DATA_BLOCK DB 811
TITLE =
AUTHOR : CB
STRUCT
WORD0 : WORD;	//
WORD1 : WORD;	//
END_STRUCT;
BEGIN
END_DATA_BLOCK
